FUNCTION_BLOCK PUBLIC FB_LampUpDownAdapter EXTENDS FB_Lamp
VAR
	fbLampUpDown		: FB_LampUpDown;
END_VAR

// Reduces the control value by 5 in the range of 10 to 100.
METHOD PUBLIC DimDown
IF (fbLampUpDown.nLightLevel >= 15) THEN
	fbLampUpDown.OneStepDown();
	fbLampUpDown.OneStepDown();
	fbLampUpDown.OneStepDown();
	fbLampUpDown.OneStepDown();
	fbLampUpDown.OneStepDown();
END_IF
IF (_ipObserver <> 0) THEN
	_ipObserver.Update(fbLampUpDown.nLightLevel);
END_IF
END_METHOD

// Increments the control value by 5 in the range of 10 to 100.
METHOD PUBLIC DimUp
IF (fbLampUpDown.nLightLevel <= 95) THEN	
	fbLampUpDown.OneStepUp();
	fbLampUpDown.OneStepUp();
	fbLampUpDown.OneStepUp();
	fbLampUpDown.OneStepUp();
	fbLampUpDown.OneStepUp();
END_IF
IF (_ipObserver <> 0) THEN
	_ipObserver.Update(fbLampUpDown.nLightLevel);
END_IF
END_METHOD

// Sets the control value to 0.
METHOD PUBLIC Off
IF (fbLampUpDown.nLightLevel > 0) THEN
	fbLampUpDown.OnOff();
END_IF
IF (_ipObserver <> 0) THEN
	_ipObserver.Update(fbLampUpDown.nLightLevel);
END_IF
END_METHOD

// Sets the control value to 100.
METHOD PUBLIC On
IF (fbLampUpDown.nLightLevel = 0) THEN
	fbLampUpDown.OnOff();
END_IF
IF (_ipObserver <> 0) THEN
	_ipObserver.Update(fbLampUpDown.nLightLevel);
END_IF
END_METHOD

END_FUNCTION_BLOCK

(* stored: Version 1.1.0.1, ProductVersion 3.1.4024.11
   POU FB_LampUpDownAdapter: Id {5ca69942-f3d0-4276-8ef2-8cc1c698a883}, SpecialFunc None
   Method DimDown: Id {8c4c7f5f-ad02-4e3b-97a6-e863a99be8f5}
   Method DimUp: Id {403b05bf-aacb-4c8b-8952-69cec07e41d6}
   Method Off: Id {b8b7ff35-eb11-4a8d-a9df-7efa1e97a4f1}
   Method On: Id {d1eb4880-a8ae-402a-909f-c11ffa6132c8} *)
